PROGRAM MAIN
VAR
END_VAR

GVL_Pers.testPeristent := GVL_Pers.testPeristent +10;
GVL_Non_Pers.testNonPers := GVL_Non_Pers.testNonPers +10;

END_PROGRAM

(* stored: Version 1.1.0.1, ProductVersion 3.1.4022.12
   POU MAIN: Id {f24976e0-536e-47c0-9e90-f6a02fca37e7}, SpecialFunc None *)
